{attribute 'GeneratedUsingTerminal: ELM3002-0000-0016'}
{attribute addProperty BoxType "ELM3002-0000-0016"}
{attribute addProperty Id "StatusAT %I*Status_543010BE7"}
{attribute addProperty CRC "2924134660"}
{attribute addProperty Size "7"}
TYPE PAI_Status_Channel_AE4AC104 EXTENDS InputBase_8311D824 :
STRUCT
	{attribute addProperty Name "Status"}
	Status AT %I* : Status_543010BE;
END_STRUCT
END_TYPE

(* stored: Version 1.2.0.0, ProductVersion 3.1.4024.11
   DUT PAI_Status_Channel_AE4AC104: Id {7b6b747a-80ba-4af2-85ad-14baeeeff276} *)
